FUNCTION_BLOCK T_ModuleCollectionOneNotInitialisedAllNotInitialised EXTENDS T_UnitTestBase
VAR
  list : T_SubModuleCollection(10);
  newModule, newModule2 : T_SubModuleMock; 
  actual1, actual2 : BOOL;
END_VAR

// Arrange
list.AddModule(newModule);
list.AddModule(newModule2);

//Act
newModule.dontInitialise := TRUE;
list.CyclicLogic();

//Assert
actual1 := NOT list.InitialisedAll;

assertion.AssertEquals_BOOL(TRUE, actual1, 'actual1 := NOT list.InitialisedAll');
TestFinished();

END_FUNCTION_BLOCK

(* stored: Version 1.1.0.1, ProductVersion 3.1.4024.12
   POU T_ModuleCollectionOneNotInitialisedAllNotInitialised: Id {151a2dae-4c8a-40b5-9770-c992893437ff}, SpecialFunc None *)
